FUNCTION Xor2 : BoolValue
VAR_INPUT
	value1 : BoolValue;
	value2 : BoolValue;
END_VAR
VAR
	p : POINTER TO BooleanExpression;
END_VAR

p := __NEW(BooleanExpression);

p^.Op2(
	operator := BooleanOperator.XORop,
	value1 := value1,
	value2 := value2
);

Xor2 := p^;

END_FUNCTION

(* stored: Version 1.1.0.1
   POU Xor2: Id {2a5298cc-0e96-4080-8ade-e2ae0feaf660}, SpecialFunc None *)
